TYPE ST_MCHMIPrepareScreen_00_05 :
STRUCT
	btmpValue_00_05	: BOOL;
END_STRUCT
END_TYPE

(* stored: Version 1.1.0.1
   DUT ST_MCHMIPrepareScreen_00_05: Id {2de4c065-2dba-02f6-1ae3-946f65721147} *)
